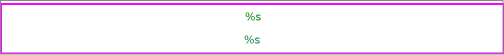
VISUALIZATION MessageBox_2  // 504x55
VAR_IN_OUT
	message_1 : ST_MessageBoxText;
	message_2 : ST_MessageBoxText;
END_VAR
    Textfield (3,2 500x30), "%s", text variable: message_1.sText
        p55702900: message_1.nColor
    Textfield (2,25 500x30), "%s", text variable: message_2.sText
        p55702900: message_2.nColor
    Rectangle (0,3 504x51)
        p3450524324: message_1.nColor
END_VISUALIZATION

(* stored: Version 1.1.0.1
   Visu MessageBox_2: Id {695357df-3db2-4a73-b9af-0569f4021190} *)
